RoboDK station: ChArUco Hand-Eye Calibration.rdk

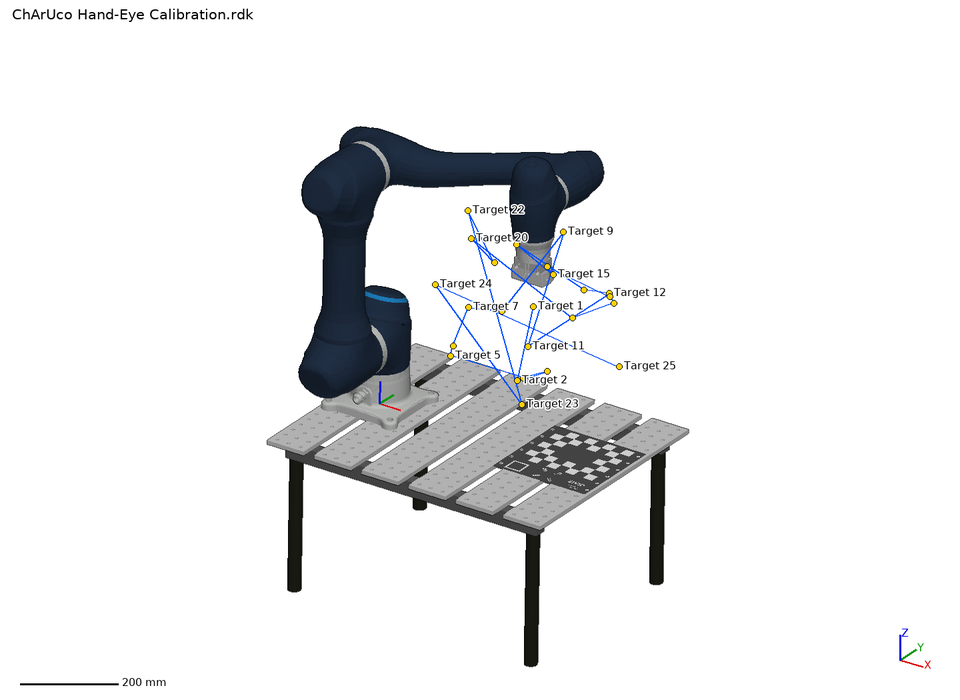
[picture v0: the station drawn from its stored meshes, robots at their saved joint values, targets as dots, program paths as lines]
Station test station (saved by RoboDK 5.9.2). Poses are relative to the parent item; angles as X-Y-Z fixed-axis rotations.
Station parameters (name, value as stored): IO_2, 0, IO_5, 1, IO_3, 0, 2, 0, 3, 0
  - program declamping (2 instructions, listed below)
  - program clamping (2 instructions, listed below)
  - frame World at (141.88, -8.76, 0) mm, rotated rx 0 ry 1.07 rz 1.07 deg
    - frame Doosan Robotics A0509 Base at (0, 0, 0) mm
      - robot Doosan Robotics A0509: 6 axes, payload 5 kg, reach 900 mm, repeatability 0.03 mm
          modified DH rows (alpha deg, a mm, theta deg, d mm): 0, 0, 0, 155.5; -90, 0, -90, 0; 0, 409, -90, 0; -90, 0, 0, 367; 90, 0, 0, 0; -90, 0, 90, 124
          base shift (0, 0, 0) mm, rotated rx 0 ry 0 rz 180 deg
          joint limits [-360, -360, -150, -360, -360, -360] to [360, 360, 150, 360, 360, 360]; home [0, 0, 90, 0, 0, 0]; saved at [-180, 0, -90, -180, 90, 180]
        - tool 560210_HGPT-35-A-B, TCP at (80, 0, 45) mm, size 42 x 50.8 x 80 mm, geometry from World
    - target Target 1 (Cartesian target) at (369.73, 0, 329.78) mm, rotated rx 180 ry -0.9 rz -180 deg; joints [0, 0.89, 90, 0, 90.005, 0] of Doosan Robotics A0509
    - target Target 2 (Cartesian target) at (444.38, -166.74, 250.05) mm, rotated rx 133.1 ry -15.8 rz 167.99 deg; joints [-36.927, 31.321, 75.186, 37.324, 105.656, -18.325] of Doosan Robotics A0509
    - target Target 3 (Cartesian target) at (473.83, -100.99, 253.33) mm, rotated rx -178.39 ry -45.91 rz 90.48 deg; joints [-28.853, 28.816, 77.201, 38.407, 99.769, 57.756] of Doosan Robotics A0509
    - target Target 4 (Cartesian target) at (424.8, -114.64, 230.02) mm, rotated rx 151.98 ry -22.98 rz 147.1 deg; joints [-29.806, 21.742, 87.221, 29.21, 92.14, 4.455] of Doosan Robotics A0509
    - target Target 5 (Cartesian target) at (294.56, -188.13, 272.14) mm, rotated rx 150.67 ry -35.8 rz 107.81 deg; joints [-56.182, 8.018, 102.133, 37.873, 95.156, 20.412] of Doosan Robotics A0509
    - target Target 6 (Cartesian target) at (247.66, -108.15, 248.22) mm, rotated rx 146.3 ry -25.62 rz 107.04 deg; joints [-56.151, -9.855, 122.018, 39.732, 83.531, 14.385] of Doosan Robotics A0509
    - target Target 7 (Cartesian target) at (227.03, -22.84, 295.09) mm, rotated rx 140.79 ry -0.03 rz 121.51 deg; joints [-43.565, -33.047, 127.08, 38.743, 77.497, 9.132] of Doosan Robotics A0509
    - target Target 8 (Cartesian target) at (275.71, 28.47, 279.93) mm, rotated rx 179.99 ry 15.94 rz -178.52 deg; joints [7.172, -21.631, 117.193, -1.661, 68.574, 6.078] of Doosan Robotics A0509
    - target Target 9 (Cartesian target) at (449.11, -12.17, 527.18) mm, rotated rx -178.96 ry -0.02 rz 161.5 deg; joints [-1.048, 23.045, 29.284, -1.256, 128, 16.683] of Doosan Robotics A0509
    - target Target 11 (Cartesian target) at (353.61, 7.9, 231.12) mm, rotated rx 179.18 ry -0.64 rz -178.49 deg; joints [0.754, 0.623, 105.904, 0.846, 74.125, -0.984] of Doosan Robotics A0509
    - target Target 12 (Cartesian target) at (421.56, 203.18, 291.56) mm, rotated rx -179.02 ry 11.76 rz 91.74 deg; joints [30.514, 17.995, 76.501, -9.814, 92.059, 119.085] of Doosan Robotics A0509
    - target Target 13 (Cartesian target) at (422.95, 105.48, 340.51) mm, rotated rx -166.84 ry -8.69 rz -172.16 deg; joints [19.802, 15.69, 72.488, -11.374, 102.8, 9.496] of Doosan Robotics A0509
    - target Target 14 (Cartesian target) at (201.07, 189.9, 344.46) mm, rotated rx 154.26 ry 15.71 rz 91.8 deg; joints [67.617, -14.808, 106.039, -29.752, 91.489, 152.133] of Doosan Robotics A0509
    - target Target 15 (Cartesian target) at (267.42, 227.11, 279.95) mm, rotated rx 153.41 ry 15.7 rz 91.8 deg; joints [59.697, -4.667, 108.23, -31.486, 76.477, 151.716] of Doosan Robotics A0509
    - target Target 16 (Cartesian target) at (313.73, 133.78, 350.06) mm, rotated rx -162.42 ry 9.67 rz -172.93 deg; joints [36.361, -4.655, 94.326, -19.989, 90.771, 30.592] of Doosan Robotics A0509
    - target Target 17 (Cartesian target) at (386.52, 257.75, 252.02) mm, rotated rx -131.78 ry -12.84 rz -159.7 deg; joints [50.116, 30.688, 76.173, -36.803, 106.82, 24.06] of Doosan Robotics A0509
    - target Target 18 (Cartesian target) at (376.48, 287.79, 221.94) mm, rotated rx -131.78 ry -12.84 rz -159.71 deg; joints [52.79, 34.417, 75.033, -34.899, 106.218, 27.798] of Doosan Robotics A0509
    - target Target 19 (Cartesian target) at (341.05, 189.95, 217.67) mm, rotated rx -160.05 ry 2.23 rz -177.13 deg; joints [39.138, 11.069, 98.699, -17.478, 81.055, 41.049] of Doosan Robotics A0509
    - target Target 20 (Cartesian target) at (95.04, 181.88, 329.99) mm, rotated rx -153.95 ry 40.94 rz 178.29 deg; joints [97.305, -9.984, 111.444, -33.669, 112.378, 105.44] of Doosan Robotics A0509
    - target Target 21 (Cartesian target) at (105.32, 254.49, 248.53) mm, rotated rx 176.56 ry 50.44 rz 150.08 deg; joints [99.326, 1.372, 116.269, -39.555, 95.462, 135.879] of Doosan Robotics A0509
    - target Target 22 (Cartesian target) at (52.31, 232.85, 360.92) mm, rotated rx 169.22 ry 39.27 rz 127.84 deg; joints [102.182, -5.557, 99.853, -28.864, 114.906, 145.039] of Doosan Robotics A0509
    - target Target 23 (Cartesian target) at (468.91, -184.56, 211.04) mm, rotated rx 159.61 ry -22.53 rz 175.62 deg; joints [-26.395, 37.366, 63.83, 11.339, 106.658, -17.352] of Doosan Robotics A0509
    - target Target 24 (Cartesian target) at (129.71, 0.01, 309.76) mm, rotated rx -180 ry 29.11 rz -180 deg; joints [0, -53.947, 125.911, 0.002, 78.925, -0.004] of Doosan Robotics A0509
    - target Target 25 (Cartesian target) at (578.97, 5.54, 251.2) mm, rotated rx 179.98 ry -30 rz -178.48 deg; joints [0.702, 53.861, 27.866, -0.496, 128.271, -1.017] of Doosan Robotics A0509
    - object Table 1200x1000mm (Welding) at (240, 0, 0) mm, size 671.5 x 542.9 x 342.9 mm, geometry from Table-1200x1000mm-Welding.sld
      - object Zivid ZVDA-CB01 Calibration Board at (103.57, -98.2, 0.2) mm, size 225 x 225 x 1.5 mm, geometry from Zivid-ZVDA-CB01-Calibration-Board.sld
  - program Prog3 (50 instructions, listed below)
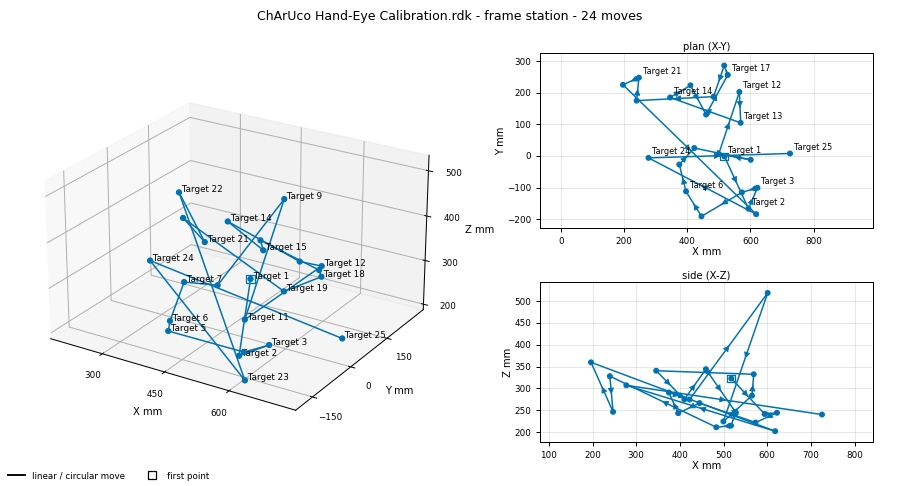
[picture p0: tool path of ChArUco Hand-Eye Calibration.rdk in frame station, 24 of 24 moves have a stored position in this frame; points joined in program order, loops and branches not executed]

--- program declamping (robot Doosan Robotics A0509) ---
  Set IO_2=1
  Set IO_2=0

--- program clamping (robot Doosan Robotics A0509) ---
  Set IO_3=1
  Set IO_3=0

--- program Prog3 (robot Doosan Robotics A0509) ---
  Set Ref.: World
  Set Tool: 560210_HGPT-35-A-B
  MoveJ (Target 1)
  Pause 2.0 s
  MoveL (Target 2)
  Pause 2.0 s
  MoveL (Target 3)
  Pause 2.0 s
  MoveL (Target 4)
  Pause 2.0 s
  MoveL (Target 5)
  Pause 2.0 s
  MoveL (Target 6)
  Pause 2.0 s
  MoveL (Target 7)
  Pause 2.0 s
  MoveL (Target 8)
  Pause 2.0 s
  MoveL (Target 9)
  Pause 2.0 s
  MoveL (Target 11)
  Pause 2.0 s
  MoveL (Target 12)
  Pause 2.0 s
  MoveL (Target 13)
  Pause 2.0 s
  MoveL (Target 14)
  Pause 2.0 s
  MoveL (Target 15)
  Pause 2.0 s
  MoveL (Target 16)
  Pause 2.0 s
  MoveL (Target 17)
  Pause 2.0 s
  MoveL (Target 18)
  Pause 2.0 s
  MoveL (Target 19)
  Pause 2.0 s
  MoveL (Target 20)
  Pause 2.0 s
  MoveL (Target 21)
  Pause 2.0 s
  MoveL (Target 22)
  Pause 2.0 s
  MoveL (Target 23)
  Pause 2.0 s
  MoveL (Target 24)
  Pause 2.0 s
  MoveL (Target 25)
  Pause 2.0 s
